// TIA Portal V18 export
TYPE "PLCtoMES_MainCheckIn"
// stored: IsFailsafeCompliant false
   STRUCT
      "P-PartIDReq" : Bool;   // PLC请求Mes标志位，MES置位M-ReqMesDone下发完成信号后，由PLC复位此信号。
      "P-PartType" : String[28];   // 产品型号 非上线工位专用，PLC读取托盘TAG工件型号MN
      "P-PartID" : Array[1..10] of String[48];   // 产品主码 下游工位读托盘或者扫码获取主工件ID，首站只给PartID，适用于上线工位要扫描主从多个零件的情况，主从工件一起和MES下发的虚拟ID绑定，如有多个主从零件码，就在P-partID[1-10]往后累加。
      "P-RecipeVer" : String[18];   // 工艺参数版本号，第一次从M-ParameterVer获取后保存
      "P-DeviceID" : Int;   // 轻量化压铸专用，压铸设备编号，机台编号，用于生成打刻数据
      "P-MoldID" : Int;   // 轻量化压铸专用，模具编号，用于生成打刻数据
      Reserve : Array[1..443] of Byte;
   END_STRUCT;
END_TYPE
